// Mitsubishi GX Works2 project: spj   PLC: Q02/Q02H

PROGRAM MAIN
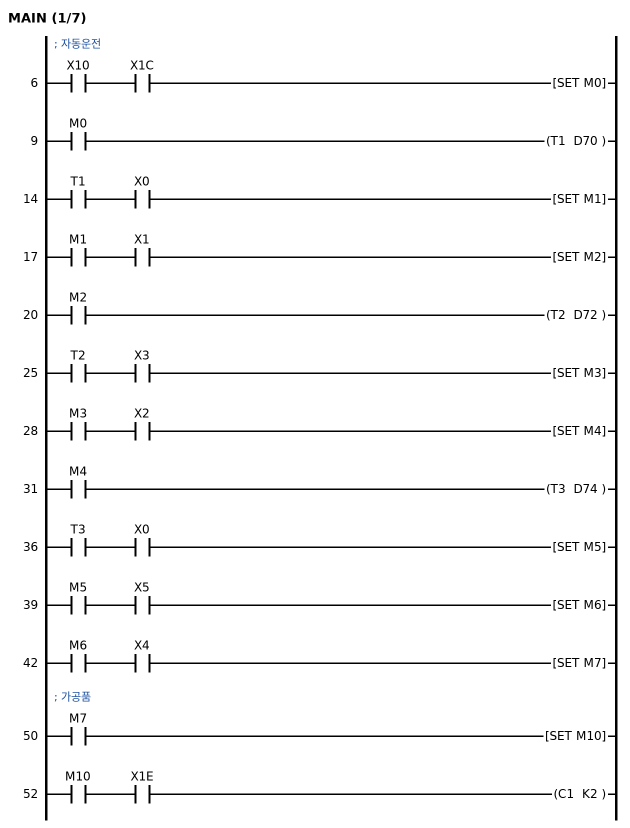
; 자동운전
6     LD      X10
      AND     X1C
      SET     M0
9     LD      M0
      OUT     T1 D70
14    LD      T1
      AND     X0
      SET     M1
17    LD      M1
      AND     X1
      SET     M2
20    LD      M2
      OUT     T2 D72
25    LD      T2
      AND     X3
      SET     M3
28    LD      M3
      AND     X2
      SET     M4
31    LD      M4
      OUT     T3 D74
36    LD      T3
      AND     X0
      SET     M5
39    LD      M5
      AND     X5
      SET     M6
42    LD      M6
      AND     X4
      SET     M7
; 가공품
50    LD      M7
      SET     M10
52    LD      M10
      AND     X1E
      OUT     C1 K2
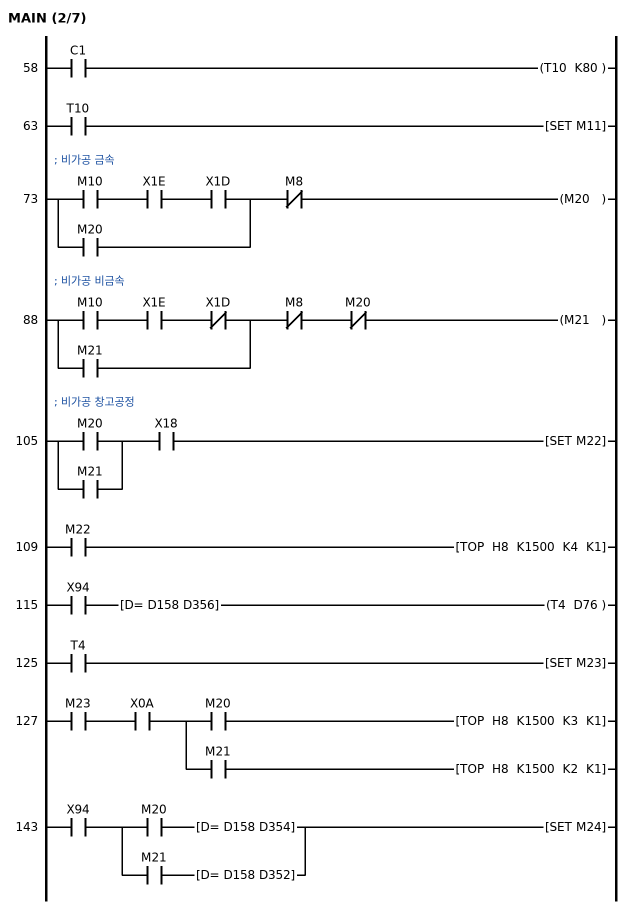
58    LD      C1
      OUT     T10 K80
63    LD      T10
      SET     M11
; 비가공 금속
73    LD      M10
      AND     X1E
      AND     X1D
      OR      M20
      ANI     M8
      OUT     M20
; 비가공 비금속
88    LD      M10
      AND     X1E
      ANI     X1D
      OR      M21
      ANI     M8
      ANI     M20
      OUT     M21
; 비가공 창고공정
105   LD      M20
      OR      M21
      AND     X18
      SET     M22
109   LD      M22
      TOP     H8 K1500 K4 K1
115   LD      X94
      ANDD=   D158 D356
      OUT     T4 D76
125   LD      T4
      SET     M23
127   LD      M23
      AND     X0A
      MPS
      AND     M20
      TOP     H8 K1500 K3 K1
      MPP
      AND     M21
      TOP     H8 K1500 K2 K1
143   LD      X94
      LD      M20
      ANDD=   D158 D354
      LD      M21
      ANDD=   D158 D352
      ORB
      ANB
      SET     M24
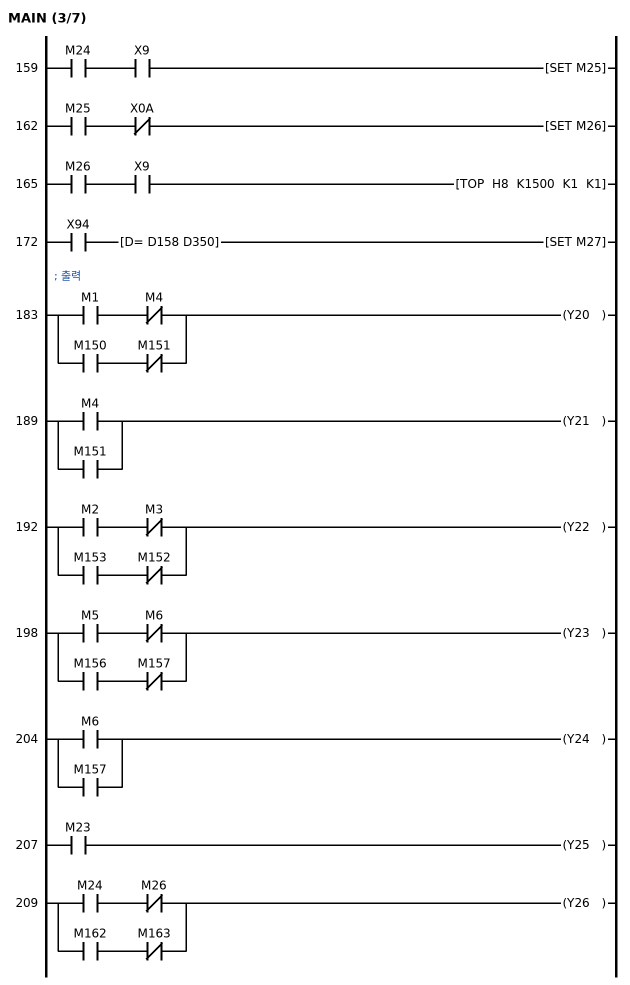
159   LD      M24
      AND     X9
      SET     M25
162   LD      M25
      ANI     X0A
      SET     M26
165   LD      M26
      AND     X9
      TOP     H8 K1500 K1 K1
172   LD      X94
      ANDD=   D158 D350
      SET     M27
; 출력
183   LD      M1
      ANI     M4
      LD      M150
      ANI     M151
      ORB
      OUT     Y20
189   LD      M4
      OR      M151
      OUT     Y21
192   LD      M2
      ANI     M3
      LD      M153
      ANI     M152
      ORB
      OUT     Y22
198   LD      M5
      ANI     M6
      LD      M156
      ANI     M157
      ORB
      OUT     Y23
204   LD      M6
      OR      M157
      OUT     Y24
207   LD      M23
      OUT     Y25
209   LD      M24
      ANI     M26
      LD      M162
      ANI     M163
      ORB
      OUT     Y26
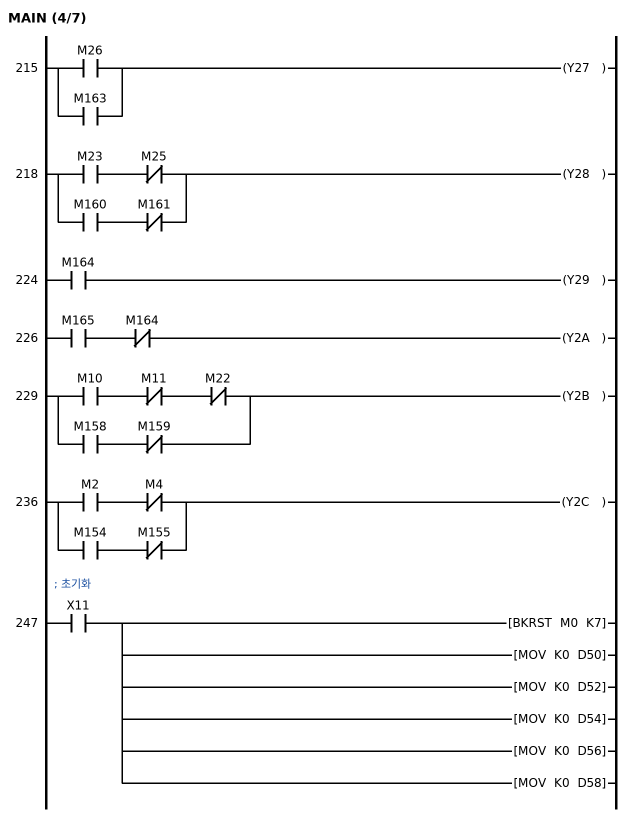
215   LD      M26
      OR      M163
      OUT     Y27
218   LD      M23
      ANI     M25
      LD      M160
      ANI     M161
      ORB
      OUT     Y28
224   LD      M164
      OUT     Y29
226   LD      M165
      ANI     M164
      OUT     Y2A
229   LD      M10
      ANI     M11
      ANI     M22
      LD      M158
      ANI     M159
      ORB
      OUT     Y2B
236   LD      M2
      ANI     M4
      LD      M154
      ANI     M155
      ORB
      OUT     Y2C
; 초기화
247   LD      X11
      BKRST   M0 K7
      MOV     K0 D50
      MOV     K0 D52
      MOV     K0 D54
      MOV     K0 D56
      MOV     K0 D58
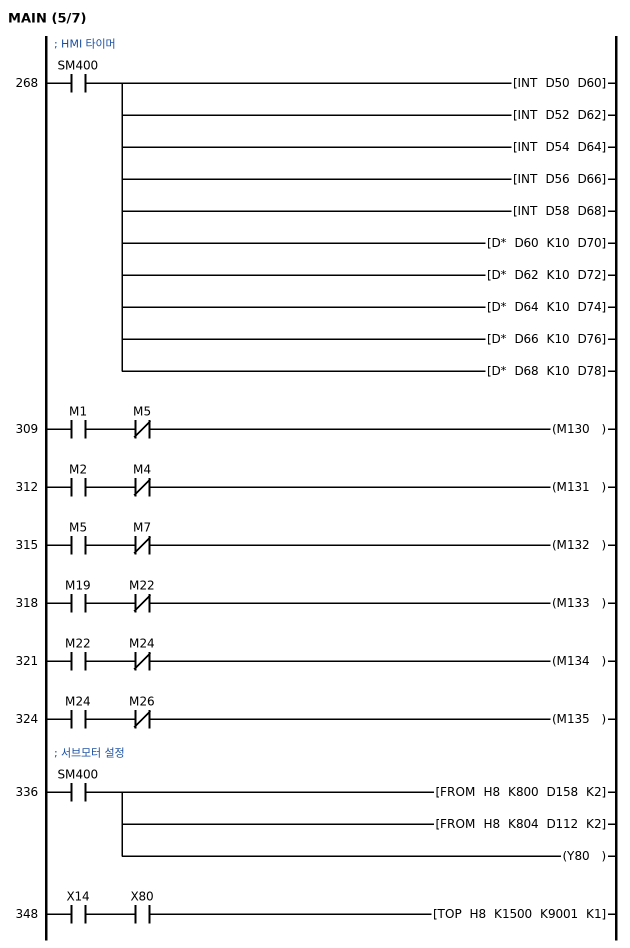
; HMI 타이머
268   LD      SM400
      INT     D50 D60
      INT     D52 D62
      INT     D54 D64
      INT     D56 D66
      INT     D58 D68
      D*      D60 K10 D70
      D*      D62 K10 D72
      D*      D64 K10 D74
      D*      D66 K10 D76
      D*      D68 K10 D78
309   LD      M1
      ANI     M5
      OUT     M130
312   LD      M2
      ANI     M4
      OUT     M131
315   LD      M5
      ANI     M7
      OUT     M132
318   LD      M19
      ANI     M22
      OUT     M133
321   LD      M22
      ANI     M24
      OUT     M134
324   LD      M24
      ANI     M26
      OUT     M135
; 서브모터 설정
336   LD      SM400
      FROM    H8 K800 D158 K2
      FROM    H8 K804 D112 K2
      OUT     Y80
348   LD      X14
      AND     X80
      TOP     H8 K1500 K9001 K1
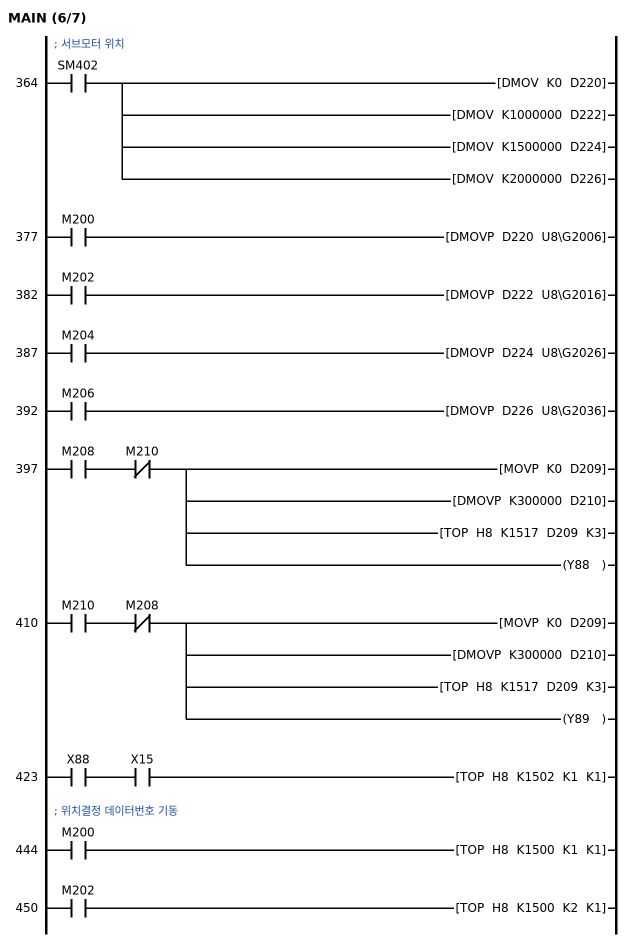
; 서브모터 위치
364   LD      SM402
      DMOV    K0 D220
      DMOV    K1000000 D222
      DMOV    K1500000 D224
      DMOV    K2000000 D226
377   LD      M200
      DMOVP   D220 U8\G2006
382   LD      M202
      DMOVP   D222 U8\G2016
387   LD      M204
      DMOVP   D224 U8\G2026
392   LD      M206
      DMOVP   D226 U8\G2036
397   LD      M208
      ANI     M210
      MOVP    K0 D209
      DMOVP   K300000 D210
      TOP     H8 K1517 D209 K3
      OUT     Y88
410   LD      M210
      ANI     M208
      MOVP    K0 D209
      DMOVP   K300000 D210
      TOP     H8 K1517 D209 K3
      OUT     Y89
423   LD      X88
      AND     X15
      TOP     H8 K1502 K1 K1
; 위치결정 데이터번호 기동
444   LD      M200
      TOP     H8 K1500 K1 K1
450   LD      M202
      TOP     H8 K1500 K2 K1
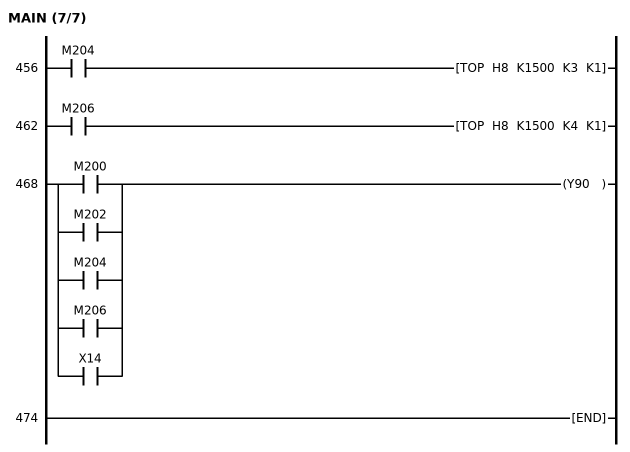
456   LD      M204
      TOP     H8 K1500 K3 K1
462   LD      M206
      TOP     H8 K1500 K4 K1
468   LD      M200
      OR      M202
      OR      M204
      OR      M206
      OR      X14
      OUT     Y90
474   END
END_PROGRAM
